TYPE (* IEC61131-3, Table 14#5 *)
  (* Standard: 1131-3 *)
  (* Version 0.0, 1/8/2024, Cheyan, Schneider Electric, Template *)
  PACKAGE Main;
  {SET_ATTRIBUTE(nxtDataType, F/ea0TupPJuJoVZpvzrlKQA4levS12OEkI6ogTkw31nr5l0edZEILHY/dfzMdMAouTKIDobrWo3b4AqhGXV9etB7pqTj5CPgZoUQ5fczaoE=)}
  AnalogueValue : STRUCT
    i : DINT;
    f : LREAL;
  END_STRUCT;
END_TYPE
